// BASE CLASS FOR EVERY UNIT/MACHINE IN THE SYSTEM
	// consists of modemanager, statemachine, UnitState interface
	// and setMode and setState methods.
	
	// UnitState interface's methods must be implemented in derived classes of UnitBaseClass
	// and MUST call this class' M_StateComplete as their last command
	
	// this function block is only meant to be run once (initialize values)
	
FUNCTION_BLOCK UnitBaseClass IMPLEMENTS ITF_UnitState
VAR_INPUT
	// input parameters for startup state and unit mode
	modeCommand	:	E_PMLProtectedUnitMode;
	command		:	E_PMLCommand;
END_VAR
VAR_OUTPUT
	currentMode		:	DINT;
	currentState	:	E_PMLState;
	initialized		:	BOOL		:= 	FALSE;
END_VAR
VAR
	
	unitModeManager		:	PML_UnitModeManager;
	stateMachine		:	PML_StateMachine;	
	wasHereSuper	:	INT	:= 	0;
END_VAR

IF (NOT initialized) THEN
	
	//enable unitmodemanager
	unitModeManager.bExecute := TRUE;
	
	// if initialization was success return true
	IF (setMode(modeCommand:=modeCommand) AND setState(command := command)) THEN
		initialized := TRUE;
	END_IF
END_IF


METHOD M_Aborted
END_METHOD

// M_Aborting is an 'acting' type state called in UnitBaseClass::setState()
// due to rising signal of emergency stop button.

// the implementation is done in derived classes
METHOD M_Aborting
M_StateComplete();
END_METHOD

{warning 'add method implementation'}
METHOD M_Clearing
M_StateComplete();
END_METHOD

{warning 'add method implementation'}
METHOD M_Complete
END_METHOD

{warning 'add method implementation'}
METHOD M_Completing
M_StateComplete();
END_METHOD

{warning 'add method implementation'}
METHOD M_Execute
END_METHOD

{warning 'add method implementation'}
METHOD M_Held
END_METHOD

{warning 'add method implementation'}
METHOD M_Holding
M_StateComplete();
END_METHOD

{warning 'add method implementation'}
METHOD M_Idle
END_METHOD

{warning 'add method implementation'}
METHOD M_Resetting
M_StateComplete();
END_METHOD

{warning 'add method implementation'}
METHOD M_Starting
M_StateComplete();
END_METHOD


// PML_StateMachine::M_StateCompleted() is what actually 
// changes the state from acting state to wait state.
// that's why this method is called after every '-ing' (acting) state.

METHOD M_StateComplete
stateMachine.M_StateComplete();
currentState := stateMachine.eState;
END_METHOD

{warning 'add method implementation'}
METHOD M_Stopped
END_METHOD

{warning 'add method implementation'}
METHOD M_Stopping
M_StateComplete();
END_METHOD

{warning 'add method implementation'}
METHOD M_Suspended
END_METHOD

{warning 'add method implementation'}
METHOD M_Suspending
M_StateComplete();
END_METHOD

{warning 'add method implementation'}
METHOD M_Undefined
END_METHOD

{warning 'add method implementation'}
METHOD M_Unholding
M_StateComplete();
END_METHOD

{warning 'add method implementation'}
METHOD M_Unsuspending
M_StateComplete();
END_METHOD

METHOD setMode : BOOL
VAR_INPUT
	modeCommand	:	DINT;
END_VAR
VAR
	prevMode	:	E_PMLProtectedUnitMode;
END_VAR
// save current mode as previous mode
prevMode := currentMode;

// update current mode
unitModeManager(eModeCommand := modeCommand, 
				eState := currentState,
				eModeStatus => currentMode);
				
// check if mode was changed, if not return false
IF(currentMode = prevMode) OR (currentMode = ePMLProtUnitMode_Invalid) THEN
	setMode := FALSE;
	RETURN;
END_IF

setMode := TRUE;
END_METHOD


// setState method. Attempts to change the state of unit according to 
// the given input command which is a result of received user signal (startButton, stopButton ... ).

(* possible commands :	
	ePMLCommand_Undefined   := 0,
	ePMLCommand_Reset       := 1,
	ePMLCommand_Start       := 2,
	ePMLCommand_Stop        := 3,
	ePMLCommand_Hold        := 4,
	ePMLCommand_Unhold      := 5,
	ePMLCommand_Suspend     := 6,
	ePMLCommand_Unsuspend   := 7,
	ePMLCommand_Abort       := 8,
	ePMLCommand_Clear       := 9
*)

METHOD setState : BOOL
VAR_INPUT
	command	:	E_PMLCommand;
END_VAR
VAR
	prevState	:	E_PMLState;	
END_VAR
wasHereSuper	:= wasHereSuper + 1;
// save current state as previous state
prevState := currentState;

// update current state
stateMachine(eMode:=currentMode, eCommand:=command, eState=>currentState);

// check whether the state was changed, if not return false
IF (currentState = prevState) OR (currentState = ePMLState_Undefined) THEN
	setState := FALSE;
	RETURN;
END_IF

setState := TRUE;

// run resulted state method.
CASE currentState OF
	
	ePMLState_Undefined:
		M_Undefined();
	
    ePMLState_Clearing:
		M_Clearing();
		
    ePMLState_Stopped:
		M_Stopped();
		
    ePMLState_Starting:
		M_Starting();
		
    ePMLState_Idle:
		M_Idle();
		
    ePMLState_Suspended:
		M_Suspended();
		
    ePMLState_Execute:
		M_Execute();
		
    ePMLState_Stopping:
		M_Stopping();
		
    ePMLState_Aborting:
		M_Aborting();
		
    ePMLState_Aborted:
		M_Aborted();
		
    ePMLState_Holding:
		M_Holding();
		
    ePMLState_Held:
		M_Held();
		
    ePMLState_Unholding:
		M_Unholding();
		
    ePMLState_Suspending:
		M_Suspending();
		
    ePMLState_Unsuspending:
		M_Unsuspending();
		
    ePMLState_Resetting:
		M_Resetting();
		
    ePMLState_Completing:
		M_Completing();
		
    ePMLState_Complete:
		M_Complete();
		
END_CASE
END_METHOD

END_FUNCTION_BLOCK

(* stored: Version 1.1.0.1, ProductVersion 3.1.4022.16
   POU UnitBaseClass: Id {aeb6491f-b3ec-42f8-9416-1e872ebf9f16}, SpecialFunc None
   Method M_Aborted: Id {997c4508-d824-4ccb-92c7-e4b4e83ad8e2}
   Method M_Aborting: Id {a2cab866-18ab-4c9f-aeb9-c9ff213eaeb6}
   Method M_Clearing: Id {5a749b99-c3ec-4cf4-ab18-53664f2d3c57}
   Method M_Complete: Id {76cf367f-98e3-4f00-83f6-5769137b65bb}
   Method M_Completing: Id {78e8f8f9-ab57-4e3f-87f0-12cd71f50a99}
   Method M_Execute: Id {6d32e3b0-53a6-4d94-a000-39c1f1969c06}
   Method M_Held: Id {18859718-e822-41fd-8bf8-24e252ff5705}
   Method M_Holding: Id {66dc536e-543c-4dee-baaf-e266bc29ac19}
   Method M_Idle: Id {3c447920-8f82-4329-ac21-183fdac9bac6}
   Method M_Resetting: Id {0e63659c-91b5-4ac9-960a-4290e83bba6d}
   Method M_Starting: Id {0e8572ed-7889-4440-9c77-d48046bbb65a}
   Method M_StateComplete: Id {a5711707-f478-4de0-8048-bf66597864d5}
   Method M_Stopped: Id {5642a46b-167d-4c98-ba93-28ffdb6b987a}
   Method M_Stopping: Id {679d777b-9988-4d27-8f5e-b6dafa5ed1b2}
   Method M_Suspended: Id {26b8c5db-c8b7-4d74-b505-1be26ec27b4f}
   Method M_Suspending: Id {b46f7b58-5421-43f5-be83-a525fe1292c9}
   Method M_Undefined: Id {3d18d60d-4641-4a9e-9873-889667e8c9d6}
   Method M_Unholding: Id {76f1bc42-e0c3-4882-9776-963356027530}
   Method M_Unsuspending: Id {7e1f4aa9-a082-4c68-a8b2-237274d1d344}
   Method setMode: Id {00f6f159-0a01-4f23-adfc-9258cf4fd8f7}
   Method setState: Id {29595849-60fa-4f5d-9eec-19649e04e713} *)
